ABB RobotStudio station: 6640_station_regular_20220308-140523.rsstn

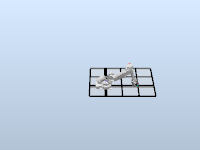
Station Station (saved by RobotStudio 21.4.9700.0)
Controller 6640_regular
  mechanical unit ROB_1: IRB6640_180_255__04, 6 joints, base frame (0, 0, 0) mm
Layout (positions relative to the parent item):
  - IRB6640_180_255__04 [mechanism, from Robots\IRB6640_180_255_G_04.rslib] at (0, 0, 0) mm; joint values [-0.014, 1.1246, 0.148, 0.7784, -1.6826, 2.9645] (rad or m)
